// TIA Portal V18 export
// export: Created 2026-06-11T05:34:05.3660526Z, ExportSetting WithDefaults, DisplayName Totally Integrated Automation Portal, DisplayVersion V18, DisplayName TIA Portal Openness, DisplayVersion V18, DisplayName TIA Portal Version Control Interface, DisplayVersion V18, DisplayName STEP 7 Professional, DisplayVersion V18, DisplayName STEP 7 Safety, DisplayVersion V18, DisplayName WinCC Professional, DisplayVersion V18
Screen "Screen_1"  1920x1080, Number=1
  ScreenLayer 
    GraphicView "Graphic view_1" at 0,0 size 1920x1080  Picture=scadabai1_1
    Circle "Circle_1" at 20,151 size 31x31
      RangeAppearanceAnimation "RangeAppearanceAnimation"
        tag 1500S_Trang_Thai
        0..0: back #ffffff, fore #000000
        1..1: back #00ff00, fore #000000
    Circle "Circle_2" at 21,426 size 30x30
      RangeAppearanceAnimation "RangeAppearanceAnimation"
        tag 1404T_Trang_Thai
        0..0: back #ffffff, fore #000000
        1..1: back #00ff00, fore #000000
    Circle "Circle_3" at 130,553 size 31x31
      RangeAppearanceAnimation "RangeAppearanceAnimation"
        tag CR_2013_FO_104_Trang_Thai
        0..0: back #ffffff, fore #000000
        1..1: back #00ff00, fore #000000
    Circle "Circle_4" at 20,751 size 32x32
      RangeAppearanceAnimation "RangeAppearanceAnimation"
        tag BFOC_SS_20_06_Trang_Thai
        0..0: back #ffffff, fore #000000
        1..1: back #00ff00, fore #000000
    IOField "I/O field_1" at 1653,536 size 71x26  DataFormat=Decimal, FormatPattern=99.9, Mode=InOutput
      ProcessValue := 1400_TT32_PV
    IOField "I/O field_2" at 651,766 size 72x23  DataFormat=Decimal, FormatPattern=99.9, Mode=InOutput
      ProcessValue := 1400_FS51_PV
    IOField "I/O field_3" at 124,828 size 99x20  DataFormat=Decimal, FormatPattern=999.9, Mode=InOutput
      ProcessValue := 1400_LGFE01_PV
    IOField "I/O field_4" at 805,697 size 74x24  DataFormat=Decimal, FormatPattern=99.9, Mode=InOutput
      ProcessValue := 1406_TX35_PV
    IOField "I/O field_7" at 741,327 size 73x20  DataFormat=Decimal, FormatPattern=999.9, Mode=InOutput
      ProcessValue := 1400_FT101_PV
    IOField "I/O field_8" at 481,270 size 76x24  DataFormat=Decimal, FormatPattern=999.9, Mode=InOutput
      ProcessValue := 1400_FT115_PV
    IOField "I/O field_9" at 1189,265 size 76x26  DataFormat=Decimal, FormatPattern=999.9, Mode=InOutput
      ProcessValue := 1400_1_02_PV
    IOField "I/O field_10" at 1201,887 size 76x25  DataFormat=Decimal, FormatPattern=999.9, Mode=InOutput
      ProcessValue := 1400_FY301_PV
    IOField "I/O field_11" at 1385,537 size 72x23  DataFormat=Decimal, FormatPattern=99.9, Mode=InOutput
      ProcessValue := 1400_TT64_PV
    Circle "Circle_6" at 946,385 size 31x31
      RangeAppearanceAnimation "RangeAppearanceAnimation"
        tag 1400_PT91_Chay
        0..0: back #ffffff, fore #000000
        1..1: back #00ff00, fore #000000
    Circle "Circle_7" at 1756,553 size 31x31
      RangeAppearanceAnimation "RangeAppearanceAnimation"
        tag PC03010T01_Trang_Thai
        0..0: back #ffffff, fore #000000
        1..1: back #00ff00, fore #000000
    Circle "Circle_8" at 1713,676 size 31x31
      RangeAppearanceAnimation "RangeAppearanceAnimation"
        tag 1401_Trang_Thai
        0..0: back #ffffff, fore #000000
        1..1: back #00ff00, fore #000000
    TextField "Text_field_Unit_I_O_field_1" at 1732,536 size 40x26  Text="<body><p>°C</p></body>"
    TextField "Text_field_Unit_I_O_field_2" at 731,766 size 40x23  Text="<body><p>Hz</p></body>"
    TextField "Text_field_Unit_I_O_field_3" at 231,828 size 40x20  Text="<body><p>%</p></body>"
    TextField "Text_field_Unit_I_O_field_4" at 887,697 size 40x24  Text="<body><p>bar</p></body>"
    TextField "Text_field_Unit_I_O_field_7" at 822,327 size 40x20  Text="<body><p>L/h</p></body>"
    TextField "Text_field_Unit_I_O_field_8" at 565,270 size 40x24  Text="<body><p>L/h</p></body>"
    TextField "Text_field_Unit_I_O_field_9" at 1273,265 size 40x26  Text="<body><p>L/h</p></body>"
    TextField "Text_field_Unit_I_O_field_10" at 1285,887 size 40x25  Text="<body><p>%</p></body>"
    TextField "Text_field_Unit_I_O_field_11" at 1465,537 size 40x23  Text="<body><p>°C</p></body>"
    Button "Btn_Login" at 1720,70 size 80x26  TextOff="<body><p>Login</p></body>"
      on Click: ShowLogonDialog()
    Button "Btn_Logout" at 1810,70 size 80x26  TextOff="<body><p>Logout</p></body>"
      on Click: Logoff()
